{attribute 'GeneratedUsingTerminal: EL1262-0000-0002'}
{attribute addProperty BoxType "EL1262-0000-0002"}
{attribute addProperty Id "Ch2_CycleCountAT %I*UINT2"}
{attribute addProperty CRC "2540327349"}
{attribute addProperty Size "2"}
TYPE Ch2_CycleCount_976A51B5 EXTENDS InputBase_8311D824 :
STRUCT
	{attribute addProperty Name "Ch2_CycleCount"}
	Ch2_CycleCount AT %I* : UINT;
END_STRUCT
END_TYPE

(* stored: Version 1.2.0.0, ProductVersion 3.1.4024.11
   DUT Ch2_CycleCount_976A51B5: Id {40844367-5b18-4363-b01b-db29ac16e447} *)
